FUNCTION_BLOCK PoolReload (* Service Interface Block to reload/update the object pool during runtime *)
  (* Standard: ISO 11783-6; Description: Copyright (c) 2025 Meisterschulen am Ostbahnhof This program and the accompanying materials are made available under the terms of the Eclipse Public License 2.0 which is available at https://www.eclipse.org/legal/epl-2.0/ SPDX-License-Identifier: EPL-2.0 Service Interface Block to reload/update the object pool during runtime This block wraps the functionality of VTC_PoolReload() from the ISOBUS driver samples. It allows reloading or updating the object pool on the VT while the application is running. The block performs the following steps: 1. Loads the pool data from the configured file (e.g., pools/pool_de.iop) 2. Opens the pool for the specified color depth 3. Calls IsoVtcPoolUpdate() to update the pool on the VT 4. Optionally applies ID range mode settings for pool manipulation Typical use cases: - Language switching during runtime - Dynamic pool updates based on application state - Reloading modified pool files Note: The pool file path is typically read from configuration. Default path: pools/pool_de.iop (German language variant) *)
  (* Version 1.0, 2025-02-27, Generated, Meisterschulen am Ostbahnhof *)
  PACKAGE isobus::UT;
  IMPORT eclipse4diac::core::TypeHash;
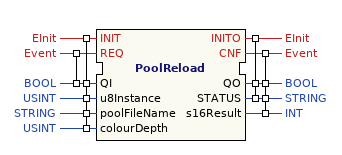
  EVENT_INPUT
    INIT : EInit WITH QI, u8Instance, poolFileName, colourDepth; (* Service Initialization *)
    REQ WITH QI; (* Service Request - Reload pool *)
  END_EVENT
  EVENT_OUTPUT
    INITO : EInit WITH QO, STATUS; (* Initialization Confirm *)
    CNF WITH QO, STATUS, s16Result; (* Confirmation - Pool reload completed *)
  END_EVENT
  VAR_INPUT
    QI : BOOL; (* Quality Input - TRUE to enable service *)
    u8Instance : USINT; (* Identifier of the VT client instance (0-255) *)
    poolFileName : STRING; (* Path to pool file (e.g., pools/pool_de.iop) *)
    colourDepth : USINT := 2; (* Color depth: 0=monochrome, 1=16 colors, 2=256 colors *)
  END_VAR
  VAR_OUTPUT
    QO : BOOL; (* Quality Output - TRUE if pool reload was successful *)
    STATUS : STRING; (* Service Status *)
    s16Result : INT; (* Return value: 0=E_NO_ERR (success), negative=error code *)
  END_VAR
END_FUNCTION_BLOCK
